Omron Sysmac Studio project conect_hmi_weintek_nx1p2 (Sysmac Studio 1.45.1.64010, StandardProject)

# Controller new_Controller_0: NX1P2-9024DT version 1.40
Units and slaves: Node86 : NX-ECC201 (E001); Unit 1 : NX-OD5121 (N1); Unit 2 : NX-OD4256 (N2); Unit 3 : NX-ID5342 (N3); Unit 4 : NX-ID5442 (N4); Node1 : GX-ID1611+OD16 (E002)
Task PrimaryTask (priority 4, period or condition 2000): Program0

VAR_GLOBAL
    start_hmi : BOOL;  (* published *)
    stop_hmi : BOOL;  (* published *)
    dong_co : BOOL;  (* at BuiltInIO://cpu/#0/Output_Bit_00; published *)
    ID5442_IN_0 : BOOL;  (* NX_ECC201_ID5442; at ECAT://node#[86,4]/Input Bit 16 bits/Input Bit 00; published *)
    ID5442_IN_1 : BOOL;  (* NX_ECC201_ID5442; at ECAT://node#[86,4]/Input Bit 16 bits/Input Bit 01; published *)
    ID5442_IN_2 : BOOL;  (* NX_ECC201_ID5442; at ECAT://node#[86,4]/Input Bit 16 bits/Input Bit 02; published *)
    ID5442_IN_3 : BOOL;  (* NX_ECC201_ID5442; at ECAT://node#[86,4]/Input Bit 16 bits/Input Bit 03; published *)
    ID5442_IN_4 : BOOL;  (* NX_ECC201_ID5442; at ECAT://node#[86,4]/Input Bit 16 bits/Input Bit 04; published *)
    ID5442_IN_5 : BOOL;  (* NX_ECC201_ID5442; at ECAT://node#[86,4]/Input Bit 16 bits/Input Bit 05; published *)
    ID5442_IN_6 : BOOL;  (* NX_ECC201_ID5442; at ECAT://node#[86,4]/Input Bit 16 bits/Input Bit 06; published *)
    ID5442_IN_7 : BOOL;  (* NX_ECC201_ID5442; at ECAT://node#[86,4]/Input Bit 16 bits/Input Bit 07; published *)
    ID5442_IN_8 : BOOL;  (* NX_ECC201_ID5442; at ECAT://node#[86,4]/Input Bit 16 bits/Input Bit 08; published *)
    ID5442_IN_9 : BOOL;  (* NX_ECC201_ID5442; at ECAT://node#[86,4]/Input Bit 16 bits/Input Bit 09; published *)
    ID5442_IN_10 : BOOL;  (* NX_ECC201_ID5442; at ECAT://node#[86,4]/Input Bit 16 bits/Input Bit 10; published *)
    ID5442_IN_11 : BOOL;  (* NX_ECC201_ID5442; at ECAT://node#[86,4]/Input Bit 16 bits/Input Bit 11; published *)
    ID5442_IN_12 : BOOL;  (* NX_ECC201_ID5442; at ECAT://node#[86,4]/Input Bit 16 bits/Input Bit 12; published *)
    ID5442_IN_13 : BOOL;  (* NX_ECC201_ID5442; at ECAT://node#[86,4]/Input Bit 16 bits/Input Bit 13; published *)
    ID5442_IN_14 : BOOL;  (* NX_ECC201_ID5442; at ECAT://node#[86,4]/Input Bit 16 bits/Input Bit 14; published *)
    ID5442_IN_15 : BOOL;  (* NX_ECC201_ID5442; at ECAT://node#[86,4]/Input Bit 16 bits/Input Bit 15; published *)
    ID5342_IN_0 : BOOL;  (* NX_ECCC201_ID5342; at ECAT://node#[86,3]/Input Bit 16 bits/Input Bit 00; published *)
    ID5342_IN_1 : BOOL;  (* NX_ECCC201_ID5342; at ECAT://node#[86,3]/Input Bit 16 bits/Input Bit 01; published *)
    ID5342_IN_2 : BOOL;  (* NX_ECCC201_ID5342; at ECAT://node#[86,3]/Input Bit 16 bits/Input Bit 02; published *)
    ID5342_IN_3 : BOOL;  (* NX_ECCC201_ID5342; at ECAT://node#[86,3]/Input Bit 16 bits/Input Bit 03; published *)
    ID5342_IN_4 : BOOL;  (* NX_ECCC201_ID5342; at ECAT://node#[86,3]/Input Bit 16 bits/Input Bit 04; published *)
    ID5342_IN_5 : BOOL;  (* NX_ECCC201_ID5342; at ECAT://node#[86,3]/Input Bit 16 bits/Input Bit 05; published *)
    ID5342_IN_6 : BOOL;  (* NX_ECCC201_ID5342; at ECAT://node#[86,3]/Input Bit 16 bits/Input Bit 06; published *)
    ID5342_IN_7 : BOOL;  (* NX_ECCC201_ID5342; at ECAT://node#[86,3]/Input Bit 16 bits/Input Bit 07; published *)
    ID5342_IN_8 : BOOL;  (* NX_ECCC201_ID5342; at ECAT://node#[86,3]/Input Bit 16 bits/Input Bit 08; published *)
    ID5342_IN_9 : BOOL;  (* NX_ECCC201_ID5342; at ECAT://node#[86,3]/Input Bit 16 bits/Input Bit 09; published *)
    ID5342_IN_10 : BOOL;  (* NX_ECCC201_ID5342; at ECAT://node#[86,3]/Input Bit 16 bits/Input Bit 10; published *)
    ID5342_IN_11 : BOOL;  (* NX_ECCC201_ID5342; at ECAT://node#[86,3]/Input Bit 16 bits/Input Bit 11; published *)
    ID5342_IN_12 : BOOL;  (* NX_ECCC201_ID5342; at ECAT://node#[86,3]/Input Bit 16 bits/Input Bit 12; published *)
    ID5342_IN_13 : BOOL;  (* NX_ECCC201_ID5342; at ECAT://node#[86,3]/Input Bit 16 bits/Input Bit 13; published *)
    ID5342_IN_14 : BOOL;  (* NX_ECCC201_ID5342; at ECAT://node#[86,3]/Input Bit 16 bits/Input Bit 14; published *)
    ID5342_IN_15 : BOOL;  (* NX_ECCC201_ID5342; at ECAT://node#[86,3]/Input Bit 16 bits/Input Bit 15; published *)
    NX1P2_IN_0 : BOOL;  (* IN_NX1P2_9024DT; at BuiltInIO://cpu/#0/Input_Bit_00; published *)
    NX1P2_IN_1 : BOOL;  (* IN_NX1P2_9024DT; at BuiltInIO://cpu/#0/Input_Bit_01; published *)
    NX1P2_IN_2 : BOOL;  (* IN_NX1P2_9024DT; at BuiltInIO://cpu/#0/Input_Bit_02; published *)
    NX1P2_IN_3 : BOOL;  (* IN_NX1P2_9024DT; at BuiltInIO://cpu/#0/Input_Bit_03; published *)
    NX1P2_IN_4 : BOOL;  (* IN_NX1P2_9024DT; at BuiltInIO://cpu/#0/Input_Bit_04; published *)
    NX1P2_IN_5 : BOOL;  (* IN_NX1P2_9024DT; at BuiltInIO://cpu/#0/Input_Bit_05; published *)
    NX1P2_IN_6 : BOOL;  (* IN_NX1P2_9024DT; at BuiltInIO://cpu/#0/Input_Bit_06; published *)
    NX1P2_IN_7 : BOOL;  (* IN_NX1P2_9024DT; at BuiltInIO://cpu/#0/Input_Bit_07; published *)
    NX1P2_IN_8 : BOOL;  (* IN_NX1P2_9024DT; at BuiltInIO://cpu/#0/Input_Bit_08; published *)
    NX1P2_IN_9 : BOOL;  (* IN_NX1P2_9024DT; at BuiltInIO://cpu/#0/Input_Bit_09; published *)
    NX1P2_IN_10 : BOOL;  (* IN_NX1P2_9024DT; at BuiltInIO://cpu/#0/Input_Bit_10; published *)
    NX1P2_IN_11 : BOOL;  (* IN_NX1P2_9024DT; at BuiltInIO://cpu/#0/Input_Bit_11; published *)
    NX1P2_IN_12 : BOOL;  (* IN_NX1P2_9024DT; at BuiltInIO://cpu/#0/Input_Bit_12; published *)
    GX_OUT_0 : BOOL;  (* GX_OUT *)
    GX_OUT_1 : BOOL;  (* GX_OUT *)
    GX_OUT_2 : BOOL;  (* GX_OUT *)
    GX_OUT_3 : BOOL;  (* GX_OUT *)
    GX_OUT_4 : BOOL;  (* GX_OUT *)
    GX_OUT_5 : BOOL;  (* GX_OUT *)
    GX_OUT_6 : BOOL;  (* GX_OUT *)
    GX_OUT_7 : BOOL;  (* GX_OUT *)
    GX_OUT_8 : BOOL;  (* GX_OUT *)
    GX_OUT_9 : BOOL;  (* GX_OUT *)
    GX_OUT_10 : BOOL;  (* GX_OUT *)
    GX_OUT_11 : BOOL;  (* GX_OUT *)
    GX_OUT_12 : BOOL;  (* GX_OUT *)
    GX_OUT_13 : BOOL;  (* GX_OUT *)
    GX_OUT_14 : BOOL;  (* GX_OUT *)
    GX_OUT_15 : BOOL;  (* GX_OUT *)
    REGISTER_GX_OUT : WORD;  (* GX_OUT; at ECAT://node#1/Write output 1st word; published *)
    NX1P2_IN_13 : BOOL;  (* IN_NX1P2_9024DT; at BuiltInIO://cpu/#0/Input_Bit_13; published *)
    REGISTER_ID5342 : WORD;  (* NX_ECCC201_ID5342; at ECAT://node#[86,3]/Input Bit 16 bits; published *)
    REGISTER_ID5442 : WORD;  (* NX_ECC201_ID5442; at ECAT://node#[86,4]/Input Bit 16 bits; published *)
    IN_GX_0 : BOOL;  (* IN_GX_ID1611; at ECAT://node#1/Read input 1st word/In Bit00; published *)
    IN_GX_1 : BOOL;  (* IN_GX_ID1611; at ECAT://node#1/Read input 1st word/In Bit01; published *)
    IN_GX_2 : BOOL;  (* IN_GX_ID1611; at ECAT://node#1/Read input 1st word/In Bit02; published *)
    IN_GX_3 : BOOL;  (* IN_GX_ID1611; at ECAT://node#1/Read input 1st word/In Bit03; published *)
    IN_GX_4 : BOOL;  (* IN_GX_ID1611; at ECAT://node#1/Read input 1st word/In Bit04; published *)
    IN_GX_5 : BOOL;  (* IN_GX_ID1611; at ECAT://node#1/Read input 1st word/In Bit05; published *)
    IN_GX_6 : BOOL;  (* IN_GX_ID1611; at ECAT://node#1/Read input 1st word/In Bit06; published *)
    IN_GX_7 : BOOL;  (* IN_GX_ID1611; at ECAT://node#1/Read input 1st word/In Bit07; published *)
    IN_GX_8 : BOOL;  (* IN_GX_ID1611; at ECAT://node#1/Read input 1st word/In Bit08; published *)
    IN_GX_9 : BOOL;  (* IN_GX_ID1611; at ECAT://node#1/Read input 1st word/In Bit09; published *)
    IN_GX_10 : BOOL;  (* IN_GX_ID1611; at ECAT://node#1/Read input 1st word/In Bit10; published *)
    IN_GX_11 : BOOL;  (* IN_GX_ID1611; at ECAT://node#1/Read input 1st word/In Bit11; published *)
    IN_GX_12 : BOOL;  (* IN_GX_ID1611; at ECAT://node#1/Read input 1st word/In Bit12; published *)
    IN_GX_13 : BOOL;  (* IN_GX_ID1611; at ECAT://node#1/Read input 1st word/In Bit13; published *)
    IN_GX_14 : BOOL;  (* IN_GX_ID1611; at ECAT://node#1/Read input 1st word/In Bit14; published *)
    IN_GX_15 : BOOL;  (* IN_GX_ID1611; at ECAT://node#1/Read input 1st word/In Bit15; published *)
    REGISTER_IN_GX : WORD;  (* IN_GX_ID1611; at ECAT://node#1/Read input 1st word; published *)
    DONG_CO_A1 : BOOL;  (* at BuiltInIO://cpu/#0/Output_Bit_01; published *)
    DONG_CO_A2 : BOOL;  (* at BuiltInIO://cpu/#0/Output_Bit_02; published *)
    START_HMI_2 : BOOL;  (* published *)
    STOP_HMI_2 : BOOL;  (* published *)
    OD4256_REGISTER : BYTE;  (* at ECAT://node#[86,2]/Output Bit 8 bits; published *)
    OD5121_REGISTER : WORD;  (* at ECAT://node#[86,1]/Output Bit 16 bits; published *)
END_VAR

PROGRAM Program0
VAR
    M0 : BOOL;
    T1 : TON;
    T2 : TON;
    VALUE_TA1 : TIME;
END_VAR
VAR_EXTERNAL
    start_hmi : BOOL;
    dong_co : BOOL;
    stop_hmi : BOOL;
    START_HMI_2 : BOOL;
    STOP_HMI_2 : BOOL;
    DONG_CO_A1 : BOOL;
    DONG_CO_A2 : BOOL;
END_VAR
VAR
    _p1 : BOOL;
END_VAR

(* Section Section0: ladder, written here as Structured Text *)

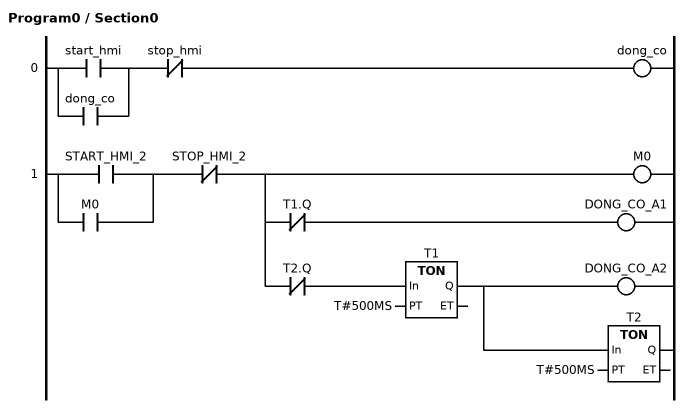
(* Rung 0 *)
dong_co := (start_hmi OR dong_co) AND NOT stop_hmi;
(* Rung 1 *)
_p1 := (START_HMI_2 OR M0) AND NOT STOP_HMI_2;
M0 := _p1;
DONG_CO_A1 := _p1 AND NOT T1.Q;
T1(In := _p1 AND NOT T2.Q, PT := T#500MS);
DONG_CO_A2 := T1.Q;
T2(In := T1.Q, PT := T#500MS);
END_PROGRAM